// TIA Portal V18 export
TYPE "IAI Par Struct"
   STRUCT
      AxisID : Int;   // 周代码
      PositionWidth : Real;   // 位置宽度
      PosCode : Int;   // 位置代码
      PushDir : Int;   // 推压方向：1,正向 2，反向
      PushWidth : Real;   // 推压宽度
      PushCurrent : Int;   // 推压电流
      TargetPosition : Array[0..49] of Real;   // 目标位置
      GoPosInterfere : Array[0..99] of Bool;   // 目标位置干涉
      Speed : Int;   // 速度
      Acceleration : Int;   // 加速度
      ChgSpeed : Int;   // 切换速度
      PushSpeed : Int;   // 压装速度
      WritePosition : Real;   // 写入位置值
      AlarmTime : Time;   // 报警时间
   END_STRUCT;
END_TYPE
